FUNCTION_BLOCK BasicFb1 (* Basic Function Block Type *)
  (* Standard: 61499-2 *)
  (* Version 0.0, 3/17/2024, linkwise-linn, LOYTEC electronics GmbH, Template *)
  PACKAGE Main;
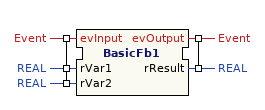
  EVENT_INPUT
    evInput WITH rVar1, rVar2; (* Initialization Request *)
  END_EVENT
  EVENT_OUTPUT
    evOutput WITH rResult; (* Execution Confirmation *)
  END_EVENT
  VAR_INPUT
    rVar1 : REAL; (* Input event qualifier *)
    rVar2 : REAL;
  END_VAR
  VAR_OUTPUT
    rResult : REAL; (* Output event qualifier *)
  END_VAR
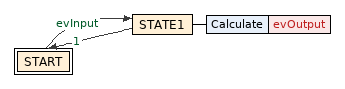
  EC_STATES
    START; (* Initial State *)
    STATE1 : Calculate -> evOutput;
  END_STATES
  EC_TRANSITIONS
    START TO STATE1 := evInput;
    STATE1 TO START := 1;
  END_TRANSITIONS
  ALGORITHM Calculate IN ST:
rResult := rVar1 + rVar2;
  END_ALGORITHM
END_FUNCTION_BLOCK
